(* IEC 61131-3 sources: xPLCCore/codesys_code/Application/COMM_FBs/FB_TcpMsgPakServer, 2 files *)

(* ---- FB_TcpMsgPakServer.st ---- *)
FUNCTION_BLOCK FB_TcpMsgPakServer
VAR_INPUT
    // --- Configuration Inputs ---
    IP_ADDRESS              : NBS.IIPAddress;  // IP Address for the server to listen on.
    PORT                    : UINT;             // Port number for the server to listen on.
    ENABLE                  : BOOL;             // Master switch to enable/disable the server.

    // --- Control Input ---
    PKT_ALLOW_NEXT          : BOOL;             // Set to TRUE to acknowledge processing of the current packet and allow the FB to provide the next one.
    // External force-reset request: caller (TCP_MSGPAK_Server) raises this
    // for one cycle when it observes sustained TX stall (xActive=TRUE but
    // Send keeps failing past TX_STALL_DROP_THRESHOLD head-drops). The
    // RX-side idle watchdog only fires on RX silence, so a half-open TX
    // path with ongoing client RX would otherwise never trigger a reset.
    xForceReset             : BOOL;
END_VAR

VAR_OUTPUT
    // --- Status and Data Outputs ---
    CLIENT                  : NBS.TCP_Connection; // The active TCP connection object. Provides access to status like xActive, xError, etc.
    PKT_IDX                 : UDINT;              // Increments each time a complete data packet is found. BUFFER_PTR and BUFFER_LEN are valid.
    BUFFER_PTR              : POINTER TO BYTE;    // Pointer to the start of the available data packet. 0 (NULL) if no data is available.
    BUFFER_LEN              : UDINT;              // Length of the available data packet in bytes. 0 if no data is available.
    // Mirrors internal xResetConnection. Caller (TCP_MSGPAK_Server) reads
    // this to suppress Send() during the 20ms grace period: once we've
    // decided to reset, xActive may still be TRUE for a few cycles, and
    // continuing to Write into an about-to-die socket either succeeds-then-
    // loses-the-reply (client never sees it, but ConsumeTail already ran)
    // or fails and bumps the stall counter for no reason.
    xResetting              : BOOL;
    // TRUE while the underlying NBS.TCP_Server has a non-null itfServer
    // (i.e. the listen-side is up). Surfaced so GET_DIAG can publish
    // it as `server_active` for external bind-health diagnostics.
    xServerActive           : BOOL;
END_VAR

VAR CONSTANT
    MAX_BUFFER_SIZE         : UDINT := 2048;
    NO_CLIENT_TIMEOUT       : TIME  := T#30S;  // Fires ServerLongIdleCount once per active-no-client window. Diagnostic for config-drift detection (bind IP wrong, firewall block); see GVL.ServerLongIdleCount comment.
END_VAR

VAR
    // --- Server and Connection Function Blocks ---
    fbServer                : NBS.TCP_Server;
    itfServer               : NBS.IServer;
    // xServerActive moved to VAR_OUTPUT above (caller / GET_DIAG read it).
    xEnableConnection       : BOOL;               // Controls the xEnable input of the TCP_Connection FB.

    // --- Data Buffers and Parsing ---
    udiBytesReceived        : UDINT;
    eReadErrorID            : NBS.ERROR;
    aInternalBuffer         : ARRAY [0..MAX_BUFFER_SIZE-1] OF BYTE;
    fbDataBuffer            : FB_DataBuffer;
    fbMsgPakParser          : FB_MsgPakLevelParser;

    // --- Connection Reset State ---
    xResetConnection        : BOOL := FALSE;      // Flag to initiate a connection reset process.
    xLastConnectionActive   : BOOL := FALSE;      // Holds CLIENT.xActive from the previous cycle.
    fbResetDelayTimer       : Standard.TON;       // Grace-period delay before tearing down the connection.
    fbIdleWatchdog          : Standard.TON;       // Fires if no bytes are received within IDLE_TIMEOUT (silent disconnect detection).
    fbNoClientTimer         : Standard.TON;       // Fires once per active-but-no-client window; drives GVL.ServerLongIdleCount.
    xLongIdleFired          : BOOL := FALSE;      // One-shot latch so fbNoClientTimer.Q only bumps the counter once per window; cleared when a client connects.

    iProcessedPacketLen     : DINT;               // Byte length of the packet currently exposed on outputs.
    iParseIdx               : DINT;               // Index of the next unparsed byte in the data buffer.

    // --- Internal Helpers ---
    tmpParserPtr            : POINTER TO BYTE;
    pre_stack_size          : DINT;
    bFirstCycle             : BOOL := TRUE;

    // --- Debug Counters ---
    DBG_recvCount           : DINT := 0;
    DBG_pktPopCount         : DINT := 0;
END_VAR
(* =========== IMPLEMENTATION =========== *)

//==================================================================================================
// FB IMPLEMENTATION
//==================================================================================================

// --- 1. First Cycle Initialization ---
IF bFirstCycle THEN
    fbMsgPakParser.ResetParser();
    iParseIdx := 0;
    fbDataBuffer.ResetBuffer(ADR(aInternalBuffer[0]), SIZEOF(aInternalBuffer));
    bFirstCycle := FALSE;
END_IF

// --- 2. Run the TCP server ---
fbServer(
    itfIPAddress      := IP_ADDRESS,
    uiPort            := PORT,
    xEnable           := ENABLE,
    udiMaxConnections := 1
);
itfServer     := fbServer.itfServer;
xServerActive := itfServer <> 0;

// --- 3. Detect connection loss or error (triggers reset) ---
IF (xLastConnectionActive AND NOT CLIENT.xActive) OR CLIENT.xError THEN
    xResetConnection := TRUE;
END_IF

// --- 3a. Rising-edge: new client connected. Bump the diagnostic counter
// so external tools can tell "the bind is healthy and someone reached
// us" from "the FSM looks healthy but nobody's actually connected".
IF NOT xLastConnectionActive AND CLIENT.xActive THEN
    GVL.ClientConnectCount := GVL.ClientConnectCount + 1;
    xLongIdleFired := FALSE;
END_IF

// --- 3b. Long-idle detector: server bound + listening but no client for
// NO_CLIENT_TIMEOUT. Bumps once per idle window (xLongIdleFired latches
// after the first Q until a client connects). Sustained growth while
// UiPingCount stays 0 means the bind is up but nobody can reach us
// (firewall, wrong port, IP mismatch on the client side, etc).
fbNoClientTimer(IN := xServerActive AND NOT CLIENT.xActive AND NOT xLongIdleFired, PT := NO_CLIENT_TIMEOUT);
IF fbNoClientTimer.Q THEN
    GVL.ServerLongIdleCount := GVL.ServerLongIdleCount + 1;
    xLongIdleFired := TRUE;
END_IF

// External force-reset (TX-side half-open detection lives in the caller;
// it raises xForceReset once it has accumulated enough head-drops to
// declare the socket dead). Counted separately from idle/read/parser
// resets via GVL.TxStallResetCount.
IF xForceReset AND NOT xResetConnection THEN
    xResetConnection := TRUE;
    GVL.TxStallResetCount := GVL.TxStallResetCount + 1;
END_IF

// Idle watchdog -- detects silent disconnections (cable unplug, client crash
// without RST, frozen renderer). The timer is fed whenever bytes arrive.
// If IDLE_TIMEOUT elapses with the socket still reporting xActive=TRUE,
// force a reset so the single-connection slot is released for the next host.
// The timeout is GVL.HostIdleTimeoutMs (>= 2 s; the UI pings every 1 s).
// The reset drops CLIENT.xActive, which runs AxisGroupSM's disconnect
// cleanup; motion already accepted runs to its end.
fbIdleWatchdog(IN := CLIENT.xActive AND NOT xResetConnection,
               PT := DINT_TO_TIME(MAX(GVL.HostIdleTimeoutMs, 2000)));
IF fbIdleWatchdog.Q AND NOT xResetConnection THEN
    xResetConnection := TRUE;
    GVL.IdleResetCount := GVL.IdleResetCount + 1;
END_IF

// --- 4. Connection reset state machine ---
// Phase 1 (delay):  20ms grace period — keep connection alive, clear stale outputs.
// Phase 2 (flush):  Disable CLIENT, flush buffers, wait for TCP stack to confirm closure.
// Phase 3 (done):   xActive dropped — clear flag, next cycle re-enables the connection.
IF xResetConnection THEN
    fbResetDelayTimer(IN := TRUE, PT := T#20MS);
    // Clear packet outputs and parser state immediately so no stale data is exposed.
    PKT_IDX    := 0;
    BUFFER_PTR := 0;
    BUFFER_LEN := 0;
    iParseIdx  := 0;
    DBG_recvCount   := 0;
    DBG_pktPopCount := 0;
    IF fbResetDelayTimer.Q THEN
        // Grace period elapsed — disable CLIENT and flush internal buffers.
        xEnableConnection := FALSE;
        fbMsgPakParser.ResetParser();
        fbDataBuffer.Clear();
        // TCP stack has confirmed the socket is closed; ready to accept a new connection.
        IF NOT CLIENT.xActive THEN
            xResetConnection := FALSE;
        END_IF
    ELSE
        xEnableConnection := xServerActive; // Still within grace period.
    END_IF
ELSE
    fbResetDelayTimer(IN := FALSE);
    xEnableConnection := xServerActive;
END_IF

// --- 5. Run the TCP connection ---
CLIENT(itfServer := itfServer, xEnable := xEnableConnection);

// --- 6. Consume the previously exposed packet from the buffer ---
IF iProcessedPacketLen > 0 THEN
    fbDataBuffer.MoveLeft(iProcessedPacketLen);
    iParseIdx           := iParseIdx - iProcessedPacketLen;
    iProcessedPacketLen := 0;
END_IF

// --- 7a. Read incoming data UNCONDITIONALLY (decoupled from PKT_ALLOW_NEXT).
// Pre-fix this read was gated by PKT_ALLOW_NEXT, so when the upstream ring
// (minfo_buf, 6 slots) backed up the socket stopped being drained AND the
// idle watchdog stopped getting fed -> IDLE_TIMEOUT(7s) tripped a spurious
// reset even though the client was healthy and still sending. Post-fix the
// socket drains into the 2KB fbDataBuffer regardless of upstream readiness,
// so the watchdog keeps getting fed as long as bytes arrive. The OS TCP
// receive buffer + 2KB app buffer give ~3-4s of headroom at 25pkt/s before
// any backpressure-driven idle reset can fire.
IF CLIENT.xActive AND fbDataBuffer.GetSpace() > 0 THEN
    eReadErrorID := CLIENT.Read(
        fbDataBuffer.GetHead(),
        fbDataBuffer.GetSpace(),
        udiCount => udiBytesReceived
    );
    // PENDING means "nothing to read yet". CODESYS Control Win returns it
    // on every idle read (Intewell returns NO_ERROR), so treating it as
    // an error reset each connection right after accept (2026-09-25).
    IF eReadErrorID <> NBS.ERROR.NO_ERROR AND eReadErrorID <> NBS.ERROR.PENDING THEN
        IF NOT xResetConnection THEN
            GVL.ReadErrorResetCount := GVL.ReadErrorResetCount + 1;
        END_IF;
        xResetConnection := TRUE;
    ELSIF udiBytesReceived > 0 THEN
        fbIdleWatchdog(IN := FALSE);  // Feed the watchdog — connection is alive.
        DBG_recvCount := DBG_recvCount + udiBytesReceived;
        fbDataBuffer.WriteLength(udiBytesReceived);
    END_IF
END_IF

// --- 7b. Parse buffered bytes (gated by PKT_ALLOW_NEXT so we only expose
// a packet when the caller has ring headroom). Buffer keeps accumulating
// across cycles while PKT_ALLOW_NEXT=FALSE -- this is the whole point of
// the read/parse split above.
IF PKT_ALLOW_NEXT AND iParseIdx < fbDataBuffer.Size() THEN
    tmpParserPtr := fbDataBuffer.GetBuffer();
    FOR iParseIdx := iParseIdx TO fbDataBuffer.Size() - 1 DO
        pre_stack_size := fbMsgPakParser.ui_level_stack_size;
        fbMsgPakParser(in_byte := tmpParserPtr[iParseIdx]);

        IF fbMsgPakParser.e_error <> E_MsgPakLevelParser_ERROR.NONE THEN
            IF NOT xResetConnection THEN
                GVL.ParserErrorResetCount := GVL.ParserErrorResetCount + 1;
            END_IF;
            xResetConnection := TRUE;
            EXIT;
        END_IF

        // Parser returned to root level — a complete packet has been assembled.
        IF pre_stack_size <> 0 AND fbMsgPakParser.ui_level_stack_size = 0 THEN
            iProcessedPacketLen := iParseIdx + 1;
            IF iProcessedPacketLen < 2 THEN
                xResetConnection := TRUE;
                EXIT;
            END_IF
            BUFFER_PTR := tmpParserPtr;
            BUFFER_LEN := DINT_TO_UDINT(iProcessedPacketLen);
            PKT_IDX    := PKT_IDX + 1;
            iParseIdx  := iParseIdx + 1;
            EXIT;
        END_IF
    END_FOR
END_IF

// --- 8. Mirror internal reset flag to the caller and update prev-cycle state.
xResetting := xResetConnection;
xLastConnectionActive := CLIENT.xActive;

(* ---- Send.st ---- *)
METHOD Send : BOOL
VAR_INPUT
	BUFFER_PTR              : POINTER TO BYTE;
	BUFFER_LEN              : UDINT;
END_VAR
VAR

    eServerTxErrorID : NBS.ERROR;
END_VAR
(* =========== IMPLEMENTATION =========== *)

Send := FALSE;
IF (CLIENT.xActive = FALSE) THEN
	RETURN;
END_IF

// 2026-06-23 code-review note: NBS.TCP_Connection.Write returns an
// ERROR enum but no bytes-sent output. We trust that NO_ERROR means
// "queued for send to the OS socket buffer" and rely on NBS / kernel
// backpressure to drop the connection on real send failure (eServerTx
// will return a non-NO_ERROR code on the NEXT call).
// If partial-send becomes a real concern (e.g. on multi-KB replies
// under heavy backpressure) we'd need an external watchdog
// (LastSendStartMs vs ack timeout) since the NBS API doesn't expose
// the actual byte count.
eServerTxErrorID := CLIENT.Write((BUFFER_PTR), BUFFER_LEN);

IF (eServerTxErrorID = TCP.ERROR.NO_ERROR) THEN
	Send := TRUE;
END_IF
